// TIA Portal V20 export
FUNCTION_BLOCK "RegisterServer"   // FB30, LAD
{ S7_Optimized_Access := 'TRUE' }
VERSION : 0.1
// stored: AutoNumber true, IsIECCheckEnabled false, SetENOAutomatically false
   VAR_INPUT
      clear : Bool;
   END_VAR
   VAR RETAIN
      NodeTable : Array[1..2] of Struct
         NodeAddr : Array[1..4] of Byte;
         NodeId : UInt;
      END_STRUCT;
   END_VAR
   VAR
      Server : MB_SERVER;
   END_VAR
   VAR RETAIN
      Link { S7_SetPoint := 'True'} : TCON_IP_v4;
   END_VAR
   VAR
      HoldReg : Array[1..4] of Int;
   END_VAR
   // NodeTable[1].NodeAddr[1] := 16#C0;
   // NodeTable[1].NodeAddr[2] := 16#A8;
   // NodeTable[1].NodeAddr[3] := 16#01;
   // NodeTable[1].NodeAddr[4] := 16#0B;
   // NodeTable[2].NodeAddr[1] := 16#C0;
   // NodeTable[2].NodeAddr[2] := 16#A8;
   // NodeTable[2].NodeAddr[3] := 16#01;
   // NodeTable[2].NodeAddr[4] := 16#0C;
   // NodeTable[1].NodeId := 1;
   // NodeTable[2].NodeId := 2;
   // Link.InterfaceId := 64;
   // Link.ID := 16#0001;
   // Link.ConnectionType := 16#0B;
   // Link.RemoteAddress.ADDR[1] := 16#C0;
   // Link.RemoteAddress.ADDR[2] := 16#A8;
   // Link.RemoteAddress.ADDR[3] := 16#01;
   // Link.RemoteAddress.ADDR[4] := 16#0A;
   // Link.RemotePort := 502;
   // HoldReg[1] := 11;
   // HoldReg[4] := -101;
BEGIN

REGION Network 1: Register server
   // Serve holding registers to the line controller.
   // Second line of the note.
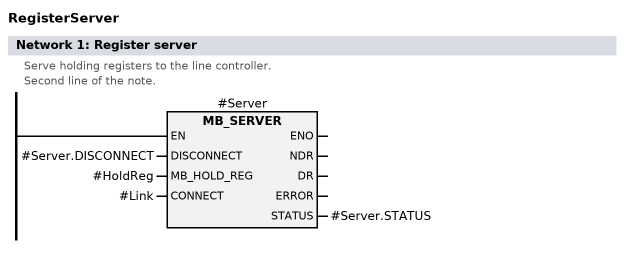
   RUNG wire#powerrail
      #Server.MB_SERVER(DISCONNECT := #Server.DISCONNECT, MB_HOLD_REG := #HoldReg, CONNECT := #Link, NDR =>, DR =>, ERROR =>, STATUS => #Server.STATUS)
   END_RUNG
   // the same network as SCL:
   #Server(DISCONNECT := #Server.DISCONNECT,   // MB_SERVER
           MB_HOLD_REG := #HoldReg,
           CONNECT := #Link,
           STATUS => #Server.STATUS);
END_REGION
END_FUNCTION_BLOCK
